FUNCTION_BLOCK CountToJob EXTENDS Job
VAR_INPUT
END_VAR
VAR_OUTPUT
END_VAR
VAR
	_nCounter: USINT;
	_nCountTo: USINT;
END_VAR

PROPERTY CountTo : USINT
GET
_nCountTo := CountTo;
END_GET
SET
IF State = JobState.Idle THEN
	_nCountTo := CountTo;
END_IF
END_SET
END_PROPERTY

(*
Executed when this job runs.  
*)
METHOD PROTECTED OnRun
_nCounter := _nCOunter + 1;
IF _nCounter >= _nCountTo THEN
	Done();
END_IF
END_METHOD

(*
Executed when this job is started.  
*)
METHOD PROTECTED OnStart
_nCounter := 0;
END_METHOD

END_FUNCTION_BLOCK

(* stored: Version 1.1.0.1
   POU CountToJob: Id {ed82a04e-7602-40f3-be4b-fa2713f6fd57}, SpecialFunc None
   Property CountTo: Id {da3c9f62-e9f4-4e95-b663-cefe7095d757}
   Get Get: Id {c8aba6a8-7048-4e1c-ae5b-5900a158522c}
   Set Set: Id {8003cf11-2b0d-4147-bdd8-0d1bbba164fc}
   Method OnRun: Id {9cd8f8e1-2d5e-4349-9f8c-55cfaeeebc5c}
   Method OnStart: Id {ad180122-f44f-45b1-8477-0eb7d514d42e} *)
